PROGRAM MAIN
VAR
	Machine		 : FB_Machine := (Name := 'Machine');
	InitComplete : BOOL;
END_VAR

IF NOT InitComplete THEN
	InitComplete := Initialize();
	RETURN;
END_IF

//Machine Cyclic Logic
Machine.CyclicLogic();

METHOD Initialize : BOOL
VAR_INPUT
END_VAR
Initialize := TRUE;
END_METHOD

END_PROGRAM

(* stored: Version 1.1.0.1, ProductVersion 3.1.4024.12
   POU MAIN: Id {f5be6099-6b61-4d94-a8d9-c23081d561a8}, SpecialFunc None
   Method Initialize: Id {ab59481b-99a0-4d4e-a6a3-d8accde04322} *)
